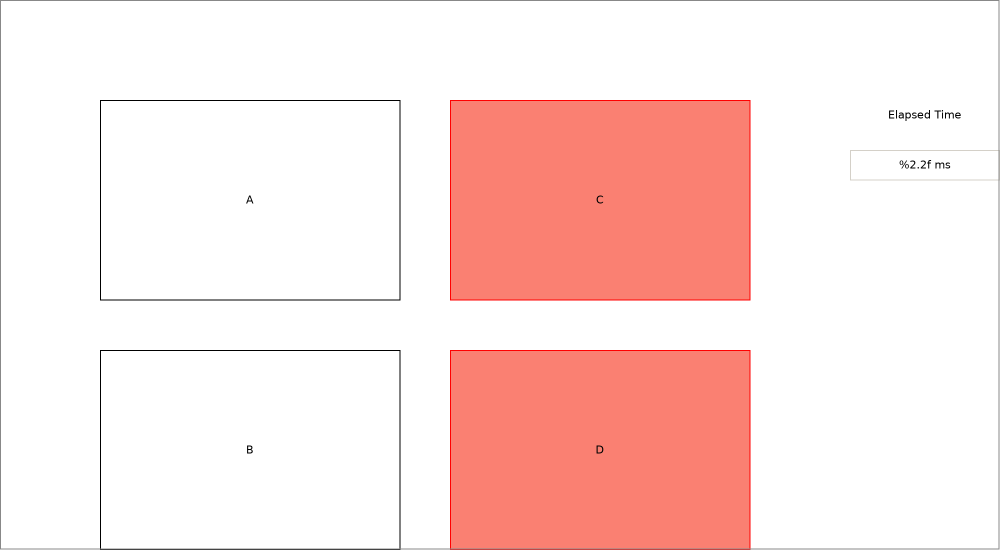
VISUALIZATION Visualization  // 1000x550
    RoundedRectangle (100,100 300x200), "A"
        OnMouseDown: toggle POU.A
    RoundedRectangle (100,350 300x200), "B"
        OnMouseDown: toggle POU.B
    RoundedRectangle (450,100 300x200), "C", colour toggle: POU.C
    RoundedRectangle (450,350 300x200), "D", colour toggle: POU.D
    Textfield (850,150 150x30), "%2.2f ms", text variable: POU.TON_0.ET
    Label (850,100 150x30), "Elapsed Time"
END_VISUALIZATION

(* stored: Version 1.1.0.1, ProductVersion 3.1.4024.3
   Visu Visualization: Id {4d5d232f-ed80-4851-94c9-f1c0a95c7db1} *)
